FUNCTION_BLOCK NVS (* Load and Store Data from NVS by Key *)
  (* Standard: 61499-2; Description: Copyright (c) 2022, 2024 HR Agrartechnik GmbH This program and the accompanying materials are made available under the terms of the Eclipse Public License 2.0 which is available at https://www.eclipse.org/legal/epl-2.0/ SPDX-License-Identifier: EPL-2.0 *)
  (* Version 1.0, 2022-09-23, Franz Höpfinger, HR Agrartechnik GmbH *)
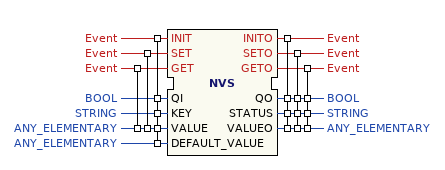
  EVENT_INPUT
    INIT WITH QI, KEY, VALUE, DEFAULT_VALUE; (* Service Initialization *)
    SET WITH VALUE; (* set value for given key *)
    GET WITH VALUE; (* get value for given key *)
  END_EVENT
  EVENT_OUTPUT
    INITO WITH QO, STATUS, VALUEO; (* Initialization Confirm *)
    SETO WITH QO, STATUS, VALUEO; (* Confirmation of SET *)
    GETO WITH QO, STATUS, VALUEO; (* Confirmation of GET *)
  END_EVENT
  VAR_INPUT
    QI : BOOL; (* Event Input Qualifier *)
    KEY : STRING; (* Key name. *)
    VALUE : ANY_ELEMENTARY; (* The value to set. *)
    DEFAULT_VALUE : ANY_ELEMENTARY; (* The value to read if there is noting in the NVS *)
  END_VAR
  VAR_OUTPUT
    QO : BOOL; (* Event Output Qualifier *)
    STATUS : STRING; (* Service Status *)
    VALUEO : ANY_ELEMENTARY; (* The output value *)
  END_VAR
END_FUNCTION_BLOCK
